PROGRAM V0_1
VAR
END_VAR

GVL.bLamp_1 := GVL.bButton_1;

END_PROGRAM

(* stored: Version 1.1.0.1, ProductVersion 3.1.4024.12
   POU V0_1: Id {eb38a907-3839-4f11-90aa-f3f66742f237}, SpecialFunc None *)
